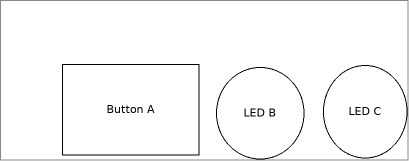
VISUALIZATION Visualization  // 409x161
    Rectangle (62,64 137x91), "Button A"
        OnMouseDown: toggle POU.A
    Ellipse (216,67 88x92), "LED B", colour toggle: POU.B
    Ellipse (323,65 84x93), "LED C", colour toggle: POU.C
END_VISUALIZATION

(* stored: Version 1.1.0.1, ProductVersion 3.1.4022.7
   Visu Visualization: Id {f9342dfc-8d06-4cb9-acb6-f3684363d463} *)
